// TwinCAT 3 PLC project sample_delivery
// Title: lcsl-plc-icl-sample-delivery
// Company: SLAC
// ProjectVersion: 0.0.0
// ProgramVersion: 3.1.4023.0
// libraries:
//   lcls-twincat-sample-delivery, * (SLAC)
//   Tc2_Standard, * (Beckhoff Automation GmbH)
//   Tc2_System, * (Beckhoff Automation GmbH)
//   Tc3_Module, * (Beckhoff Automation GmbH)
// project tree:
//   GVLs/ GVL_SDS.TcGVL
//   / PlcTask.TcTTO, SerialComm.TcTTO (not stored)
//   POUs/ MAIN.TcPOU, SerialTxRx.TcPOU
// real-time tasks:
//   TASK PlcTask: cycle T#10ms, priority 20, ADS port 350
//   TASK SerialComm: cycle T#5ms, priority 1, ADS port 351
// I/O:
//   DEVICE MAIN (EtherCAT)
// variable links:
//   sample_delivery Instance <-> MAIN (EtherCAT)/Bronkhorst MFM A
//     PlcTask Inputs/GVL_SDS.BronkhorstA.stMFM.i_rFlow <-> TxPDO Map/fMeasure
//     PlcTask Outputs/GVL_SDS.BronkhorstA.stMFM.q_rSetpoint <-> RxPDO Map/fSetpoint
//   sample_delivery Instance <-> MAIN (EtherCAT)/Bronkhorst MFM B
//     PlcTask Inputs/GVL_SDS.BronkhorstB.stMFM.i_rFlow <-> TxPDO Map/fMeasure
//     PlcTask Outputs/GVL_SDS.BronkhorstB.stMFM.q_rSetpoint <-> RxPDO Map/fSetpoint
//   sample_delivery Instance <-> MAIN (EtherCAT)/Bronkhorst MFM C
//     PlcTask Inputs/GVL_SDS.BronkhorstC.stMFM.i_rFlow <-> TxPDO Map/fMeasure
//     PlcTask Outputs/GVL_SDS.BronkhorstC.stMFM.q_rSetpoint <-> RxPDO Map/fSetpoint
//   sample_delivery Instance <-> MAIN (EtherCAT)/Bronkhorst MFM D
//     PlcTask Inputs/GVL_SDS.BronkhorstD.stMFM.i_rFlow <-> TxPDO Map/fMeasure
//     PlcTask Outputs/GVL_SDS.BronkhorstD.stMFM.q_rSetpoint <-> RxPDO Map/fSetpoint
//   sample_delivery Instance <-> MAIN (EtherCAT)/Gas_Mani (EP1111)
//     PlcTask Inputs/GVL_SDS.GasMan.stBaseIO.i_SyncUnitWC <-> WcState/WcState
//   sample_delivery Instance <-> MAIN (EtherCAT)/Gas_Mani_ValveCtrl (EP2338-0001)
//     PlcTask Outputs/GVL_SDS.GasMan.stValve[{1..7}].qxDO <-> Channel {9..15}/Output  (7 links)
//   sample_delivery Instance <-> MAIN (EtherCAT)/Gas_Mani_ValveRbk (EP2338-0001)
//     PlcTask Inputs/GVL_SDS.GasMan.stValve[{1..7}].ixOPN <-> Channel {1..7}/Input  (7 links)
//   sample_delivery Instance <-> MAIN (EtherCAT)/M3 Selector A (EP1111)
//     PlcTask Inputs/GVL_SDS.M3SelectorA.stBaseIO.i_SyncUnitWC <-> WcState/WcState
//   sample_delivery Instance <-> MAIN (EtherCAT)/M3 Selector A Digital IO (EP2338-1001)
//     PlcTask Outputs/GVL_SDS.M3SelectorA.stShaker01.q_xPwrDO <-> Channel 9/Output
//     PlcTask Outputs/GVL_SDS.M3SelectorA.stShaker02.q_xPwrDO <-> Channel 10/Output
//     PlcTask Outputs/GVL_SDS.M3SelectorA.stShaker03.q_xPwrDO <-> Channel 11/Output
//     PlcTask Outputs/GVL_SDS.M3SelectorA.stShaker04.q_xPwrDO <-> Channel 12/Output
//   sample_delivery Instance <-> MAIN (EtherCAT)/M3 Selector A Serial IO (EP6002-0002)
//     SerialComm Inputs/GVL_SDS.M3SelectorA.stSensSerial.stComIn/Status <-> COM TxPDO-Map Inputs Channel 1/Status
//     SerialComm Inputs/GVL_SDS.M3SelectorA.stViciSerial.stComIn/Status <-> COM TxPDO-Map Inputs Channel 2/Status
//     SerialComm Outputs/GVL_SDS.M3SelectorA.stSensSerial.stComOut/Ctrl <-> COM RxPDO-Map Outputs Channel 1/Ctrl
//     SerialComm Outputs/GVL_SDS.M3SelectorA.stViciSerial.stComOut/Ctrl <-> COM RxPDO-Map Outputs Channel 2/Ctrl
//   sample_delivery Instance <-> MAIN (EtherCAT)/M3 Selector B (EP1111)
//     PlcTask Inputs/GVL_SDS.M3SelectorB.stBaseIO.i_SyncUnitWC <-> WcState/WcState
//   sample_delivery Instance <-> MAIN (EtherCAT)/M3 Selector B Digital IO (EP2338-1001)
//     PlcTask Outputs/GVL_SDS.M3SelectorB.stShaker01.q_xPwrDO <-> Channel 9/Output
//     PlcTask Outputs/GVL_SDS.M3SelectorB.stShaker02.q_xPwrDO <-> Channel 10/Output
//     PlcTask Outputs/GVL_SDS.M3SelectorB.stShaker03.q_xPwrDO <-> Channel 11/Output
//     PlcTask Outputs/GVL_SDS.M3SelectorB.stShaker04.q_xPwrDO <-> Channel 12/Output
//   sample_delivery Instance <-> MAIN (EtherCAT)/M3 Selector B Serial IO (EP6002-0002)
//     SerialComm Inputs/GVL_SDS.M3SelectorB.stSensSerial.stComIn/Status <-> COM TxPDO-Map Inputs Channel 1/Status
//     SerialComm Inputs/GVL_SDS.M3SelectorB.stViciSerial.stComIn/Status <-> COM TxPDO-Map Inputs Channel 2/Status
//     SerialComm Outputs/GVL_SDS.M3SelectorB.stSensSerial.stComOut/Ctrl <-> COM RxPDO-Map Outputs Channel 1/Ctrl
//     SerialComm Outputs/GVL_SDS.M3SelectorB.stViciSerial.stComOut/Ctrl <-> COM RxPDO-Map Outputs Channel 2/Ctrl
//   sample_delivery Instance <-> MAIN (EtherCAT)/M3 Selector C (EP1111)
//     PlcTask Inputs/GVL_SDS.M3SelectorC.stBaseIO.i_SyncUnitWC <-> WcState/WcState
//   sample_delivery Instance <-> MAIN (EtherCAT)/M3 Selector C Digital IO (EP2338-1001)
//     PlcTask Outputs/GVL_SDS.M3SelectorC.stShaker01.q_xPwrDO <-> Channel 9/Output
//     PlcTask Outputs/GVL_SDS.M3SelectorC.stShaker02.q_xPwrDO <-> Channel 10/Output
//     PlcTask Outputs/GVL_SDS.M3SelectorC.stShaker03.q_xPwrDO <-> Channel 11/Output
//     PlcTask Outputs/GVL_SDS.M3SelectorC.stShaker04.q_xPwrDO <-> Channel 12/Output
//   sample_delivery Instance <-> MAIN (EtherCAT)/M3 Selector C Serial IO (EP6002-0002)
//     SerialComm Inputs/GVL_SDS.M3SelectorC.stSensSerial.stComIn/Status <-> COM TxPDO-Map Inputs Channel 1/Status
//     SerialComm Inputs/GVL_SDS.M3SelectorC.stViciSerial.stComIn/Status <-> COM TxPDO-Map Inputs Channel 2/Status
//     SerialComm Outputs/GVL_SDS.M3SelectorC.stSensSerial.stComOut/Ctrl <-> COM RxPDO-Map Outputs Channel 1/Ctrl
//     SerialComm Outputs/GVL_SDS.M3SelectorC.stViciSerial.stComOut/Ctrl <-> COM RxPDO-Map Outputs Channel 2/Ctrl
//   sample_delivery Instance <-> MAIN (EtherCAT)/M3 Selector D (EP1111)
//     PlcTask Inputs/GVL_SDS.M3SelectorD.stBaseIO.i_SyncUnitWC <-> WcState/WcState
//   sample_delivery Instance <-> MAIN (EtherCAT)/M3 Selector D Digital IO (EP2338-1001)
//     PlcTask Outputs/GVL_SDS.M3SelectorD.stShaker01.q_xPwrDO <-> Channel 9/Output
//     PlcTask Outputs/GVL_SDS.M3SelectorD.stShaker02.q_xPwrDO <-> Channel 10/Output
//     PlcTask Outputs/GVL_SDS.M3SelectorD.stShaker03.q_xPwrDO <-> Channel 11/Output
//     PlcTask Outputs/GVL_SDS.M3SelectorD.stShaker04.q_xPwrDO <-> Channel 12/Output
//   sample_delivery Instance <-> MAIN (EtherCAT)/M3 Selector D Serial IO (EP6002-0002)
//     SerialComm Inputs/GVL_SDS.M3SelectorD.stSensSerial.stComIn/Status <-> COM TxPDO-Map Inputs Channel 1/Status
//     SerialComm Inputs/GVL_SDS.M3SelectorD.stViciSerial.stComIn/Status <-> COM TxPDO-Map Inputs Channel 2/Status
//     SerialComm Outputs/GVL_SDS.M3SelectorD.stSensSerial.stComOut/Ctrl <-> COM RxPDO-Map Outputs Channel 1/Ctrl
//     SerialComm Outputs/GVL_SDS.M3SelectorD.stViciSerial.stComOut/Ctrl <-> COM RxPDO-Map Outputs Channel 2/Ctrl
//   sample_delivery Instance <-> MAIN (EtherCAT)/PCM A (EP1111)
//     PlcTask Inputs/GVL_SDS.PCMA.stBaseIO.i_SyncUnitWC <-> WcState/WcState
//   sample_delivery Instance <-> MAIN (EtherCAT)/PCM A (EP4374-0002)
//     PlcTask Inputs/GVL_SDS.PCMA.stPropAir1.i_iPressRB <-> AI Inputs Channel 1/Value
//     PlcTask Inputs/GVL_SDS.PCMA.stPropAir2.i_iPressRB <-> AI Inputs Channel 2/Value
//     PlcTask Outputs/GVL_SDS.PCMA.stPropAir1.q_iPressCt <-> AO Outputs Channel 3/Analog output
//     PlcTask Outputs/GVL_SDS.PCMA.stPropAir2.q_iPressCt <-> AO Outputs Channel 4/Analog output
//   sample_delivery Instance <-> MAIN (EtherCAT)/PCM A (EP6002-0002)
//     SerialComm Inputs/GVL_SDS.PCMA.stSerial1.stComIn/Status <-> COM TxPDO-Map Inputs Channel 1/Status
//     SerialComm Inputs/GVL_SDS.PCMA.stSerial2.stComIn/Status <-> COM TxPDO-Map Inputs Channel 2/Status
//     SerialComm Outputs/GVL_SDS.PCMA.stSerial1.stComOut/Ctrl <-> COM RxPDO-Map Outputs Channel 1/Ctrl
//     SerialComm Outputs/GVL_SDS.PCMA.stSerial2.stComOut/Ctrl <-> COM RxPDO-Map Outputs Channel 2/Ctrl
//   sample_delivery Instance <-> MAIN (EtherCAT)/PCM B (EP1111)
//     PlcTask Inputs/GVL_SDS.PCMB.stBaseIO.i_SyncUnitWC <-> WcState/WcState
//   sample_delivery Instance <-> MAIN (EtherCAT)/PCM B (EP4374-0002)
//     PlcTask Inputs/GVL_SDS.PCMB.stPropAir1.i_iPressRB <-> AI Inputs Channel 1/Value
//     PlcTask Inputs/GVL_SDS.PCMB.stPropAir2.i_iPressRB <-> AI Inputs Channel 2/Value
//     PlcTask Outputs/GVL_SDS.PCMB.stPropAir1.q_iPressCt <-> AO Outputs Channel 3/Analog output
//     PlcTask Outputs/GVL_SDS.PCMB.stPropAir2.q_iPressCt <-> AO Outputs Channel 4/Analog output
//   sample_delivery Instance <-> MAIN (EtherCAT)/PCM B (EP6002-0002)
//     SerialComm Inputs/GVL_SDS.PCMB.stSerial1.stComIn/Status <-> COM TxPDO-Map Inputs Channel 1/Status
//     SerialComm Inputs/GVL_SDS.PCMB.stSerial2.stComIn/Status <-> COM TxPDO-Map Inputs Channel 2/Status
//     SerialComm Outputs/GVL_SDS.PCMB.stSerial1.stComOut/Ctrl <-> COM RxPDO-Map Outputs Channel 1/Ctrl
//     SerialComm Outputs/GVL_SDS.PCMB.stSerial2.stComOut/Ctrl <-> COM RxPDO-Map Outputs Channel 2/Ctrl
//   sample_delivery Instance <-> MAIN (EtherCAT)/PCM C (EP1111)
//     PlcTask Inputs/GVL_SDS.PCMC.stBaseIO.i_SyncUnitWC <-> WcState/WcState
//   sample_delivery Instance <-> MAIN (EtherCAT)/PCM C (EP4374-0002)
//     PlcTask Inputs/GVL_SDS.PCMC.stPropAir1.i_iPressRB <-> AI Inputs Channel 1/Value
//     PlcTask Inputs/GVL_SDS.PCMC.stPropAir2.i_iPressRB <-> AI Inputs Channel 2/Value
//     PlcTask Outputs/GVL_SDS.PCMC.stPropAir1.q_iPressCt <-> AO Outputs Channel 3/Analog output
//     PlcTask Outputs/GVL_SDS.PCMC.stPropAir2.q_iPressCt <-> AO Outputs Channel 4/Analog output
//   sample_delivery Instance <-> MAIN (EtherCAT)/PCM C (EP6002-0002)
//     SerialComm Inputs/GVL_SDS.PCMC.stSerial1.stComIn/Status <-> COM TxPDO-Map Inputs Channel 1/Status
//     SerialComm Inputs/GVL_SDS.PCMC.stSerial2.stComIn/Status <-> COM TxPDO-Map Inputs Channel 2/Status
//     SerialComm Outputs/GVL_SDS.PCMC.stSerial1.stComOut/Ctrl <-> COM RxPDO-Map Outputs Channel 1/Ctrl
//     SerialComm Outputs/GVL_SDS.PCMC.stSerial2.stComOut/Ctrl <-> COM RxPDO-Map Outputs Channel 2/Ctrl
//   sample_delivery Instance <-> MAIN (EtherCAT)/PCM D (EP1111)
//     PlcTask Inputs/GVL_SDS.PCMD.stBaseIO.i_SyncUnitWC <-> WcState/WcState
//   sample_delivery Instance <-> MAIN (EtherCAT)/PCM D (EP4374-0002)
//     PlcTask Inputs/GVL_SDS.PCMD.stPropAir1.i_iPressRB <-> AI Inputs Channel 1/Value
//     PlcTask Inputs/GVL_SDS.PCMD.stPropAir2.i_iPressRB <-> AI Inputs Channel 2/Value
//     PlcTask Outputs/GVL_SDS.PCMD.stPropAir1.q_iPressCt <-> AO Outputs Channel 3/Analog output
//     PlcTask Outputs/GVL_SDS.PCMD.stPropAir2.q_iPressCt <-> AO Outputs Channel 4/Analog output
//   sample_delivery Instance <-> MAIN (EtherCAT)/PCM D (EP6002-0002)
//     SerialComm Inputs/GVL_SDS.PCMD.stSerial1.stComIn/Status <-> COM TxPDO-Map Inputs Channel 1/Status
//     SerialComm Inputs/GVL_SDS.PCMD.stSerial2.stComIn/Status <-> COM TxPDO-Map Inputs Channel 2/Status
//     SerialComm Outputs/GVL_SDS.PCMD.stSerial1.stComOut/Ctrl <-> COM RxPDO-Map Outputs Channel 1/Ctrl
//     SerialComm Outputs/GVL_SDS.PCMD.stSerial2.stComOut/Ctrl <-> COM RxPDO-Map Outputs Channel 2/Ctrl
//   sample_delivery Instance <-> MAIN (EtherCAT)/Solenoid Pair A Digital IO (EP2338-0001)
//     PlcTask Outputs/GVL_SDS.SolenoidPairA.q_xDO1 <-> Channel 9/Output
//     PlcTask Outputs/GVL_SDS.SolenoidPairA.q_xDO2 <-> Channel 10/Output

CONFIGURATION sample_delivery
    RESOURCE PLC ON TwinCAT3
        TASK PlcTask(INTERVAL := T#10ms, PRIORITY := 20);
        PROGRAM MAIN WITH PlcTask : MAIN;
    END_RESOURCE
END_CONFIGURATION

// ---- GVLs/GVL_SDS.TcGVL
VAR_GLOBAL
{attribute 'pytmc' := 'pv: MFX:SDS:SEL:A'}
{attribute 'TcLinkTo' := '.stSensSerial.stComIn.Status := TIIB[M3 Selector A Serial IO (EP6002-0002)]^COM TxPDO-Map Inputs Channel 1^Status;
                          .stViciSerial.stComIn.Status := TIIB[M3 Selector A Serial IO (EP6002-0002)]^COM TxPDO-Map Inputs Channel 2^Status;
                          .stSensSerial.stComOut.Ctrl := TIID^MAIN (EtherCAT)^M3 Selector A Serial IO (EP6002-0002)^COM RxPDO-Map Outputs Channel 1^Ctrl;
                          .stViciSerial.stComOut.Ctrl := TIID^MAIN (EtherCAT)^M3 Selector A Serial IO (EP6002-0002)^COM RxPDO-Map Outputs Channel 2^Ctrl;
                          .stShaker01.q_xPwrDO := TIIB[M3 Selector A Digital IO (EP2338-1001)]^Channel 9^Output;
                          .stShaker02.q_xPwrDO := TIIB[M3 Selector A Digital IO (EP2338-1001)]^Channel 10^Output;
                          .stShaker03.q_xPwrDO := TIIB[M3 Selector A Digital IO (EP2338-1001)]^Channel 11^Output;
                          .stShaker04.q_xPwrDO := TIIB[M3 Selector A Digital IO (EP2338-1001)]^Channel 12^Output;
                          .stBaseIO.i_SyncUnitWC := TIID^MAIN (EtherCAT)^M3 Selector A (EP1111)^WcState^WcState;
'}
M3SelectorA : FB_SelectorM3;

{attribute 'pytmc' := 'pv: MFX:SDS:SEL:B'}
{attribute 'TcLinkTo' := '.stSensSerial.stComIn.Status := TIIB[M3 Selector B Serial IO (EP6002-0002)]^COM TxPDO-Map Inputs Channel 1^Status;
                          .stViciSerial.stComIn.Status := TIIB[M3 Selector B Serial IO (EP6002-0002)]^COM TxPDO-Map Inputs Channel 2^Status;
                          .stSensSerial.stComOut.Ctrl := TIID^MAIN (EtherCAT)^M3 Selector B Serial IO (EP6002-0002)^COM RxPDO-Map Outputs Channel 1^Ctrl;
                          .stViciSerial.stComOut.Ctrl := TIID^MAIN (EtherCAT)^M3 Selector B Serial IO (EP6002-0002)^COM RxPDO-Map Outputs Channel 2^Ctrl;
                          .stShaker01.q_xPwrDO := TIIB[M3 Selector B Digital IO (EP2338-1001)]^Channel 9^Output;
                          .stShaker02.q_xPwrDO := TIIB[M3 Selector B Digital IO (EP2338-1001)]^Channel 10^Output;
                          .stShaker03.q_xPwrDO := TIIB[M3 Selector B Digital IO (EP2338-1001)]^Channel 11^Output;
                          .stShaker04.q_xPwrDO := TIIB[M3 Selector B Digital IO (EP2338-1001)]^Channel 12^Output;
                          .stBaseIO.i_SyncUnitWC := TIID^MAIN (EtherCAT)^M3 Selector B (EP1111)^WcState^WcState
'}
M3SelectorB : FB_SelectorM3;

{attribute 'pytmc' := 'pv: MFX:SDS:SEL:C'}
{attribute 'TcLinkTo' := '.stSensSerial.stComIn.Status := TIIB[M3 Selector C Serial IO (EP6002-0002)]^COM TxPDO-Map Inputs Channel 1^Status;
                          .stViciSerial.stComIn.Status := TIIB[M3 Selector C Serial IO (EP6002-0002)]^COM TxPDO-Map Inputs Channel 2^Status;
                          .stSensSerial.stComOut.Ctrl := TIID^MAIN (EtherCAT)^M3 Selector C Serial IO (EP6002-0002)^COM RxPDO-Map Outputs Channel 1^Ctrl;
                          .stViciSerial.stComOut.Ctrl := TIID^MAIN (EtherCAT)^M3 Selector C Serial IO (EP6002-0002)^COM RxPDO-Map Outputs Channel 2^Ctrl;
                          .stShaker01.q_xPwrDO := TIIB[M3 Selector C Digital IO (EP2338-1001)]^Channel 9^Output;
                          .stShaker02.q_xPwrDO := TIIB[M3 Selector C Digital IO (EP2338-1001)]^Channel 10^Output;
                          .stShaker03.q_xPwrDO := TIIB[M3 Selector C Digital IO (EP2338-1001)]^Channel 11^Output;
                          .stShaker04.q_xPwrDO := TIIB[M3 Selector C Digital IO (EP2338-1001)]^Channel 12^Output;
                          .stBaseIO.i_SyncUnitWC := TIID^MAIN (EtherCAT)^M3 Selector C (EP1111)^WcState^WcState
'}
M3SelectorC : FB_SelectorM3;

{attribute 'pytmc' := 'pv: MFX:SDS:SEL:D'}
{attribute 'TcLinkTo' := '.stSensSerial.stComIn.Status := TIIB[M3 Selector D Serial IO (EP6002-0002)]^COM TxPDO-Map Inputs Channel 1^Status;
                          .stViciSerial.stComIn.Status := TIIB[M3 Selector D Serial IO (EP6002-0002)]^COM TxPDO-Map Inputs Channel 2^Status;
                          .stSensSerial.stComOut.Ctrl := TIID^MAIN (EtherCAT)^M3 Selector D Serial IO (EP6002-0002)^COM RxPDO-Map Outputs Channel 1^Ctrl;
                          .stViciSerial.stComOut.Ctrl := TIID^MAIN (EtherCAT)^M3 Selector D Serial IO (EP6002-0002)^COM RxPDO-Map Outputs Channel 2^Ctrl;
                          .stShaker01.q_xPwrDO := TIIB[M3 Selector D Digital IO (EP2338-1001)]^Channel 9^Output;
                          .stShaker02.q_xPwrDO := TIIB[M3 Selector D Digital IO (EP2338-1001)]^Channel 10^Output;
                          .stShaker03.q_xPwrDO := TIIB[M3 Selector D Digital IO (EP2338-1001)]^Channel 11^Output;
                          .stShaker04.q_xPwrDO := TIIB[M3 Selector D Digital IO (EP2338-1001)]^Channel 12^Output;
                          .stBaseIO.i_SyncUnitWC := TIID^MAIN (EtherCAT)^M3 Selector D (EP1111)^WcState^WcState
'}
M3SelectorD : FB_SelectorM3;

{attribute 'pytmc' := 'pv: MFX:SDS:PCM:A'}
{attribute 'TcLinkTo' := '.stPropAir1.i_iPressRB := TIID^MAIN (EtherCAT)^PCM A (EP4374-0002)^AI Inputs Channel 1^Value;
                          .stPropAir2.i_iPressRB := TIID^MAIN (EtherCAT)^PCM A (EP4374-0002)^AI Inputs Channel 2^Value;
                          .stPropAir1.q_iPressCt := TIID^MAIN (EtherCAT)^PCM A (EP4374-0002)^AO Outputs Channel 3^Analog output;
                          .stPropAir2.q_iPressCt := TIID^MAIN (EtherCAT)^PCM A (EP4374-0002)^AO Outputs Channel 4^Analog output;
                          .stSerial1.stComIn.Status := TIID^MAIN (EtherCAT)^PCM A (EP6002-0002)^COM TxPDO-Map Inputs Channel 1^Status;
                          .stSerial2.stComIn.Status := TIID^MAIN (EtherCAT)^PCM A (EP6002-0002)^COM TxPDO-Map Inputs Channel 2^Status;
                          .stSerial1.stComOut.Ctrl := TIID^MAIN (EtherCAT)^PCM A (EP6002-0002)^COM RxPDO-Map Outputs Channel 1^Ctrl;
                          .stSerial2.stComOut.Ctrl := TIID^MAIN (EtherCAT)^PCM A (EP6002-0002)^COM RxPDO-Map Outputs Channel 2^Ctrl;
                          .stBaseIO.i_SyncUnitWC := TIID^MAIN (EtherCAT)^PCM A (EP1111)^WcState^WcState;
'}
PCMA : FB_PressureControlModule;

{attribute 'pytmc' := 'pv: MFX:SDS:PCM:B'}
{attribute 'TcLinkTo' := '.stPropAir1.i_iPressRB := TIID^MAIN (EtherCAT)^PCM B (EP4374-0002)^AI Inputs Channel 1^Value;
                          .stPropAir2.i_iPressRB := TIID^MAIN (EtherCAT)^PCM B (EP4374-0002)^AI Inputs Channel 2^Value;
                          .stPropAir1.q_iPressCt := TIID^MAIN (EtherCAT)^PCM B (EP4374-0002)^AO Outputs Channel 3^Analog output;
                          .stPropAir2.q_iPressCt := TIID^MAIN (EtherCAT)^PCM B (EP4374-0002)^AO Outputs Channel 4^Analog output;
                          .stSerial1.stComIn.Status := TIID^MAIN (EtherCAT)^PCM B (EP6002-0002)^COM TxPDO-Map Inputs Channel 1^Status;
                          .stSerial2.stComIn.Status := TIID^MAIN (EtherCAT)^PCM B (EP6002-0002)^COM TxPDO-Map Inputs Channel 2^Status;
                          .stSerial1.stComOut.Ctrl := TIID^MAIN (EtherCAT)^PCM B (EP6002-0002)^COM RxPDO-Map Outputs Channel 1^Ctrl;
                          .stSerial2.stComOut.Ctrl := TIID^MAIN (EtherCAT)^PCM B (EP6002-0002)^COM RxPDO-Map Outputs Channel 2^Ctrl;
                          .stBaseIO.i_SyncUnitWC := TIID^MAIN (EtherCAT)^PCM B (EP1111)^WcState^WcState;

'}
PCMB : FB_PressureControlModule;

{attribute 'pytmc' := 'pv: MFX:SDS:PCM:C'}
{attribute 'TcLinkTo' := '.stPropAir1.i_iPressRB := TIID^MAIN (EtherCAT)^PCM C (EP4374-0002)^AI Inputs Channel 1^Value;
                          .stPropAir2.i_iPressRB := TIID^MAIN (EtherCAT)^PCM C (EP4374-0002)^AI Inputs Channel 2^Value;
                          .stPropAir1.q_iPressCt := TIID^MAIN (EtherCAT)^PCM C (EP4374-0002)^AO Outputs Channel 3^Analog output;
                          .stPropAir2.q_iPressCt := TIID^MAIN (EtherCAT)^PCM C (EP4374-0002)^AO Outputs Channel 4^Analog output;
                          .stSerial1.stComIn.Status := TIID^MAIN (EtherCAT)^PCM C (EP6002-0002)^COM TxPDO-Map Inputs Channel 1^Status;
                          .stSerial2.stComIn.Status := TIID^MAIN (EtherCAT)^PCM C (EP6002-0002)^COM TxPDO-Map Inputs Channel 2^Status;
                          .stSerial1.stComOut.Ctrl := TIID^MAIN (EtherCAT)^PCM C (EP6002-0002)^COM RxPDO-Map Outputs Channel 1^Ctrl;
                          .stSerial2.stComOut.Ctrl := TIID^MAIN (EtherCAT)^PCM C (EP6002-0002)^COM RxPDO-Map Outputs Channel 2^Ctrl;
                          .stBaseIO.i_SyncUnitWC := TIID^MAIN (EtherCAT)^PCM C (EP1111)^WcState^WcState;
'}
PCMC : FB_PressureControlModule;

{attribute 'pytmc' := 'pv: MFX:SDS:PCM:D'}
{attribute 'TcLinkTo' := '.stPropAir1.i_iPressRB := TIID^MAIN (EtherCAT)^PCM D (EP4374-0002)^AI Inputs Channel 1^Value;
                          .stPropAir2.i_iPressRB := TIID^MAIN (EtherCAT)^PCM D (EP4374-0002)^AI Inputs Channel 2^Value;
                          .stPropAir1.q_iPressCt := TIID^MAIN (EtherCAT)^PCM D (EP4374-0002)^AO Outputs Channel 3^Analog output;
                          .stPropAir2.q_iPressCt := TIID^MAIN (EtherCAT)^PCM D (EP4374-0002)^AO Outputs Channel 4^Analog output;
                          .stSerial1.stComIn.Status := TIID^MAIN (EtherCAT)^PCM D (EP6002-0002)^COM TxPDO-Map Inputs Channel 1^Status;
                          .stSerial2.stComIn.Status := TIID^MAIN (EtherCAT)^PCM D (EP6002-0002)^COM TxPDO-Map Inputs Channel 2^Status;
                          .stSerial1.stComOut.Ctrl := TIID^MAIN (EtherCAT)^PCM D (EP6002-0002)^COM RxPDO-Map Outputs Channel 1^Ctrl;
                          .stSerial2.stComOut.Ctrl := TIID^MAIN (EtherCAT)^PCM D (EP6002-0002)^COM RxPDO-Map Outputs Channel 2^Ctrl;
                          .stBaseIO.i_SyncUnitWC := TIID^MAIN (EtherCAT)^PCM D (EP1111)^WcState^WcState;
'}
PCMD : FB_PressureControlModule;

{attribute 'pytmc' := 'pv: MFX:SDS:MAN'}
{attribute 'TcLinkTo' := '.stValve[1].qxDO := TIIB[Gas_Mani_ValveCtrl (EP2338-0001)]^Channel 9^Output;
                          .stValve[1].ixOPN := TIIB[Gas_Mani_ValveRbk (EP2338-0001)]^Channel 1^Input;
                          .stValve[2].qxDO := TIIB[Gas_Mani_ValveCtrl (EP2338-0001)]^Channel 10^Output;
                          .stValve[2].ixOPN := TIIB[Gas_Mani_ValveRbk (EP2338-0001)]^Channel 2^Input;
                          .stValve[3].qxDO := TIIB[Gas_Mani_ValveCtrl (EP2338-0001)]^Channel 11^Output;
                          .stValve[3].ixOPN := TIIB[Gas_Mani_ValveRbk (EP2338-0001)]^Channel 3^Input;
                          .stValve[4].qxDO := TIIB[Gas_Mani_ValveCtrl (EP2338-0001)]^Channel 12^Output;
                          .stValve[4].ixOPN := TIIB[Gas_Mani_ValveRbk (EP2338-0001)]^Channel 4^Input;
                          .stValve[5].qxDO := TIIB[Gas_Mani_ValveCtrl (EP2338-0001)]^Channel 13^Output;
                          .stValve[5].ixOPN := TIIB[Gas_Mani_ValveRbk (EP2338-0001)]^Channel 5^Input;
                          .stValve[6].qxDO := TIIB[Gas_Mani_ValveCtrl (EP2338-0001)]^Channel 14^Output;
                          .stValve[6].ixOPN := TIIB[Gas_Mani_ValveRbk (EP2338-0001)]^Channel 6^Input;
                          .stValve[7].qxDO := TIIB[Gas_Mani_ValveCtrl (EP2338-0001)]^Channel 15^Output;
                          .stValve[7].ixOPN := TIIB[Gas_Mani_ValveRbk (EP2338-0001)]^Channel 7^Input;
                          .stBaseIO.i_SyncUnitWC :=	TIID^MAIN (EtherCAT)^Gas_Mani (EP1111)^WcState^WcState;
'}
GasMan : FB_GasManifold;

{attribute 'pytmc' := 'pv: MFX:SDS:MFM:A'}
{attribute 'TcLinkTo' := '.stMFM.i_rFlow := TIID^MAIN (EtherCAT)^Bronkhorst MFM A^TxPDO Map^fMeasure;
                          .stMFM.q_rSetpoint := TIID^MAIN (EtherCAT)^Bronkhorst MFM A^RxPDO Map^fSetpoint;
'}
BronkhorstA : FB_BronkhorstMFM;

{attribute 'pytmc' := 'pv: MFX:SDS:MFM:B'}
{attribute 'TcLinkTo' := '.stMFM.i_rFlow := TIID^MAIN (EtherCAT)^Bronkhorst MFM B^TxPDO Map^fMeasure;
                          .stMFM.q_rSetpoint := TIID^MAIN (EtherCAT)^Bronkhorst MFM B^RxPDO Map^fSetpoint;
'}
BronkhorstB : FB_BronkhorstMFM;

{attribute 'pytmc' := 'pv: MFX:SDS:MFM:C'}
{attribute 'TcLinkTo' := '.stMFM.i_rFlow := TIID^MAIN (EtherCAT)^Bronkhorst MFM C^TxPDO Map^fMeasure;
                          .stMFM.q_rSetpoint := TIID^MAIN (EtherCAT)^Bronkhorst MFM C^RxPDO Map^fSetpoint;
'}
BronkhorstC : FB_BronkhorstMFM;

{attribute 'pytmc' := 'pv: MFX:SDS:MFM:D'}
{attribute 'TcLinkTo' := '.stMFM.i_rFlow := TIID^MAIN (EtherCAT)^Bronkhorst MFM D^TxPDO Map^fMeasure;
                          .stMFM.q_rSetpoint := TIID^MAIN (EtherCAT)^Bronkhorst MFM D^RxPDO Map^fSetpoint;
'}
BronkhorstD : FB_BronkhorstMFM;

{attribute 'pytmc' := 'pv: MFX:SDS:SPR:A'}
{attribute 'TcLinkTo' := '.q_xDO1 := TIIB[Solenoid Pair A Digital IO (EP2338-0001)]^Channel 9^Output;
                          .q_xDO2 := TIIB[Solenoid Pair A Digital IO (EP2338-0001)]^Channel 10^Output;
'}
SolenoidPairA : FB_SolenoidPair;




END_VAR

// ---- POUs/MAIN.TcPOU
PROGRAM MAIN
VAR

END_VAR

M3SelectorA();
M3SelectorB();
M3SelectorC();
M3SelectorD();
PCMA();
PCMB();
PCMC();
PCMD();
GasMan();
BronkhorstA();
BronkhorstB();
BronkhorstC();
BronkhorstD();
SolenoidPairA();

(* Following execution of all the programs, set the first pass false *)
g_xFirstPass := FALSE;

END_PROGRAM

// ---- POUs/SerialTxRx.TcPOU
PROGRAM SerialTxRx
VAR
END_VAR

M3SelectorA.SerialComm();
M3SelectorB.SerialComm();
M3SelectorC.SerialComm();
M3SelectorD.SerialComm();

PCMA.SerialComm();
PCMB.SerialComm();
PCMC.SerialComm();
PCMD.SerialComm();

END_PROGRAM
